(* Logix 5000 project; controller Reto_1 vendor 1 type 14 code 156 rev 30.11; software revision 30.00 *)

TASK MainTask (continuous, watchdog 500 ms) : MainProgram

MODULES
   Local : vendor 1 type 14 code 156 (Compact 0, rev 30.11)
      DigIN : 1769-IQ16 (Compact 4, rev 1.1, Input RPI 20 ms)
      DigOUT : vendor 1 type 7 code 86 (Compact 5, rev 2.1, Output RPI 20 ms)
END_MODULES

VAR_GLOBAL   (* controller tags *)
   Arranque_FactoryIO : BOOL;
   Arranque_Fisico : ALIAS FOR Local:4:I.Data.1;
   Banda_2 : ALIAS FOR Local:5:O.Data.6;
   Con_Compuerta : ALIAS FOR Local:5:O.Data.5;
   Contraer_D_E : BOOL;
   CTU_01 : COUNTER := (PRE := 1, ACC := 1, DN := 1);   // ¿Hay cajas en banda 2?
   CTU_02 : COUNTER := (PRE := 5, DN := 1);   // Contador de cajas
   D_IN_1 : BOOL := 1;   // Sensor 1 FactoryIO
   D_IN_2 : BOOL := 1;   // Sensor Banda 2
   D_IN_3 : BOOL;   // Boton apagado FactoryIO
   D_IN_4 : BOOL;
   D_IN_5 : BOOL := 1;   // Boton Encendido FactoryIO
   D_IN_6 : BOOL;   // Boton Reset FactoryIO
   D_OUT_4 : BOOL;   // Banda 1 FactoryIO
   D_OUT_5 : BOOL;   // Banda 2 FactoryIO
   D_OUT_6 : BOOL := 1;   // Compuerta central FactoryIO
   Ext_Compuerta : ALIAS FOR Local:5:O.Data.4;
   Extender_D_E : BOOL;
   Extender_S_E : BOOL;
   F_OUT_1 : REAL := 10.0;   // Velocidad Banda 2 FactoryIO
   INT_OUT_0 : DINT;   // Contador FactoryIO
   Motor_Fisico1 : ALIAS FOR Local:5:O.Data.0;
   Stop_FactoryIO : BOOL;
   Stop_Fisico : ALIAS FOR Local:4:I.Data.0;
   Temp : BOOL := 1;
   TIM_01 : TIMER := (PRE := 2500, EN := 1, DN := 1);
END_VAR

PROGRAM MainProgram   (* main routine MainRoutine *)

ROUTINE MainRoutine   (* ladder *)
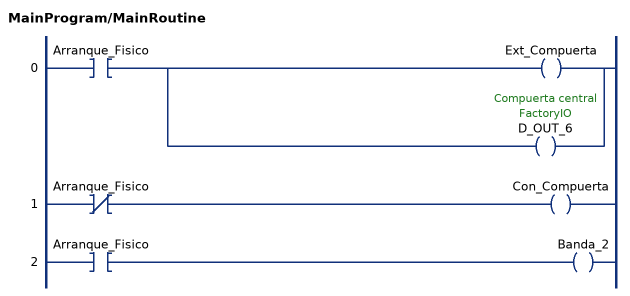
   0: XIC(Arranque_Fisico)[OTE(Ext_Compuerta) ,OTE(D_OUT_6) ];
   1: XIO(Arranque_Fisico)OTE(Con_Compuerta);
   2: XIC(Arranque_Fisico)OTE(Banda_2);
END_ROUTINE
END_PROGRAM
